Fanuc KAREL source: kt00618.KL

-- PROVISIONAL review KL for V940-1; original PC SHA256 dd81a786f4a361e70a242c2db5459bd7fe7e90efad272591928dd585a6937645
-- Incomplete behavior may be omitted. Consult companion uncertainty JSON. Do not deploy.
PROGRAM KT00618
%NOLOCKGROUP
VAR
  B1 : BOOLEAN
  B2 : BOOLEAN
  OUT : BOOLEAN
BEGIN
  B1 = TRUE
  B2 = FALSE
  B1 = TRUE
  B2 = FALSE
  OUT = NOT (B1)
END KT00618
